KUKA KRL program: TestStationMoves.src, TestStationMoves.dat

--- TestStationMoves.src ---
&ACCESS RVO
&REL 5
DEF  TestStationMoves (lnActSt :IN)
   INT lnActSt,lnUsedBase,lnUsedTool
   INT lnJobNr
   INT lnCornerNumber

   ;FOLD INIT
      CONTINUE
      ;IF ($T1 OR $T2)THEN
         GLOBAL INTERRUPT DECL 3 WHEN $STOPMESS==TRUE DO IR_STOPM ( )
         INTERRUPT ON 3
         BAS (#INITMOV,0)
         lnActSt = 2
         PTP $POS_ACT
      ;ENDIF

      PTP XHOME

      ; Used Base and tool
      lnUsedBase = 11
      lnUsedTool = 11
      gnLastToolNr = 3
      lnCornerNumber = 1

      BASE_DATA[lnUsedBase] = BASE_DATA[16]
      TOOL_DATA[lnUsedTool] = TOOL_DATA[4] :{X 0,Y 0,Z 0,A 0,B 0,C 0}
   ;ENDFOLD
   ;MoveSettings (nBase: IN, nTool: IN, nAcc: IN, nVel : IN )

   ;MoveSettings(lnUsedBase, lnUsedTool, 100, 500)
   MoveSettings(0, 1, 100, 500)
   PTP XST20_ST1_1 C_PTP
   PTP XST20_ST1_10 C_PTP

   REPEAT
      lnCornerNumber = lnCornerNumber +1
      SWITCH lnCornerNumber

         CASE 2
            BASE_DATA[lnUsedBase] = BASE_DATA[lnCornerNumber]
         CASE 3
            BASE_DATA[lnUsedBase] = BASE_DATA[lnCornerNumber]:{X 0,Y 0,Z 0,A -180,B 0,C 0}
         CASE 4
            BASE_DATA[lnUsedBase] = BASE_DATA[lnCornerNumber]:{X 0,Y 0,Z 0,A 90,B 0,C 0}
         CASE 5
            BASE_DATA[lnUsedBase] = BASE_DATA[lnCornerNumber]:{X 0,Y 0,Z 0,A 140,B 0,C 0}
       ENDSWITCH


      MoveSettings(0, 1, 100, 500)
      LIN XST1 C_VEL

      MoveSettings(lnUsedBase, lnUsedTool, 100, 500)

      LIN lfPrePos[3] C_VEL

      WAIT SEC 0.1

      MoveSettings(0, 1, 100, 500)



      LIN XST1 C_VEL


   UNTIL lnCornerNumber >= 5

   PTP XHOME

END

DEF endOfJob()
   gbJob1StartedSt[1] = FALSE
   gbJob1DoneSt[1]    = TRUE
   gnMillingCounter = gnMillingCounter+1
END

--- TestStationMoves.dat ---
&ACCESS RVO
&REL 5
DEFDAT  TestStationMoves


DECL FRAME lfPrePos[3]
lfPrePos[1]={X -150.000,Y 0.0,Z 150.000,A 0.0,B 0.0,C 0.0}
lfPrePos[2]={X 0.0,Y 0.0,Z 25.0,A 0.0,B 0.0,C 0.0}
lfPrePos[3]={X 0.0,Y 0.0,Z 150.0,A 0.0,B 0.0,C 0.0}


DECL FRAME lfWorkPos[12]
   lfWorkPos[1]={X 0,Y 0,Z 5.000,A 0.0,B 0.0,C 0.0}
   lfWorkPos[2]={X 0,Y 25.0,Z 0.0000,A 0.0,B 0.0,C 0.0}

   lfWorkPos[3]={X 1800,Y 56.0,Z 0.0000,A -73.0,B 0.0,C 0.0}
   lfWorkPos[4]={X 1695,Y 25.0,Z 0.0000,A -73.0,B 0.0,C 0.0}
   lfWorkPos[5]={X 1670,Y 1400.0,Z 0.0000,A 15.0,B 0.0,C 0.0}
   lfWorkPos[6]={X 1700,Y 1329.0,Z 0.0000,A 15.0,B 0.0,C 0.0}
   lfWorkPos[7]={X -100,Y 1305.0,Z 0.0000,A -15.0,B 0.0,C 0.0}
   lfWorkPos[8]={X 5.3,Y 1353,Z 0.0000,A -15.0,B 0.0,C 0.0}
   lfWorkPos[9]={X 30,Y -160.0,Z 0.0000,A 63.0, B 0.0,C 0.0}
   lfWorkPos[10]={X 30,Y -160.0,Z 200.0000,A 0, B 0.0,C 0.0}


   lfWorkPos[11]={X 0,Y 0.0,Z 0.0000,A 0.0,B 0.0,C 0.0}
   lfWorkPos[12]={X 0,Y 0.0,Z 0.0000,A 0.0,B 0.0,C 0.0}


ENDDAT
